(* Logix 5000 project; controller RG_Chopper vendor 1 type 14 code 235 rev 32.12; software revision 32.04; part 5 of 6 *)
(* tags used below, declared in another part *)
   CIP_CAUSTIC_RUNNING : ALIAS FOR SIGNAL_OUT_RG_CHOPPER.4;
   CYC_RUN : BOOL;   // Production Cycle Running
   DBX102_CTL : HOA_CTRL_v2;   // DBX102 Product Discharge Pump Control Block
   DBX102_FAULT : BOOL;   // DBX-102 Discharge Pump Drive Fault
   DBX102_M_FAULT : BOOL;   // DBX-102 Discharge Pump Drive or Motor Fault
   DBX102_SPD : ANLG_SCALE;   // DBX-102 Product Pump Speed Scaling
   DBX102_SPD_AM : PUSH_PUSH_PB;   // DBX-102 Speed Push-Push Button Control
   DBX102_SPD_IN : REAL;   // DBX-102 Product Pump User Requested Speed
   DBX102_SPD_OUT : REAL;   // DBX-102 VFD Alternate Requested Speed
   DBX102_SPD_PB : BOOL;   // DBX-102 Speed Auto / Manual PB
   DBX102_SPD_REQ : REAL;   // DBX-102 VFD Requested Speed
   DBX102_START : BOOL;   // DBX-102 Product Pump VFD START
   DBX102B_S_En : BOOL;   // DBX-102 Drive Safety Enable
   DBX103_AUX : BOOL;   // DBX-103 Water Pump Aux
   DBX104_CTL : HOA_CTRL_v2;   // DBX-104 Reversing Motor Starter Control
   DBX104_DWN : BOOL;   // DBX-104 Drum Dumper VFD Direction DOWN
   DBX104_FAULT : BOOL;   // DBX-104 Dumper Elevator Drive Fault
   DBX104_M_FAULT : BOOL;   // DBX-104 Dumper Elevator Drive or Motor Fault
   DBX104_S_DIR_EN : BOOL;   // DBX-104 Dump Elevator Direction Enabled
   DBX104_S_DWN : BOOL;   // DBX-104 Dump Elevator DOWN (Safety)
   DBX104_S_START : BOOL;   // DBX-104 Dump Elevator START (Safety)
   DBX104_S_UP : BOOL;   // DBX-104 Dump Elevator UP (Safety)
   DBX104_SPD : ANLG_SCALE;   // DBX-104 Product Pump Speed Scaling
   DBX104_SPD_AM : PUSH_PUSH_PB;   // DBX-104 Speed Push-Push Button Control
   DBX104_SPD_IN : DINT;   // DBX-102 Product Pump User Requested Speed
   DBX104_SPD_OUT : DINT;   // DBX-104 VFD Alternate Requested Speed
   DBX104_SPD_PB : BOOL;   // DBX-104 Speed Auto / Manual PB
   DBX104_SPD_REQ : DINT;   // DBX-104 VFD Requested Speed
   DBX104_START : BOOL;   // DBX-104 Drum Dumper VFD START
   DBX104_UP : BOOL;   // DBX-104 Drum Dumper VFD Direction UP
   DBX104B_S_En : BOOL;   // DBX-104 Drive Enable Safety
   DL101_Scl : REAL;
   DLT101_LVL_SCL : REAL;   // Tank Level Scaled (0.0 - 100.0%)
   DLT101_Tk : TK_CTRL;   // Tank Level Control
   DTT101 : REAL;   // DTT-101 Hot Water Temperature Analong In
   DWN_MKBK : BOOL;   // Elevator Down Make / Break LS_L1 Detection
   Fault_ACK : BOOL;   // Fault Acknowledge
   Gate_SW1 : DCI_MONITOR;   // Safety Switch Gate_SW1 SW105 A/B
   Gate_SW2 : DCI_MONITOR;   // Safety Switch Gate_SW2 SW108 A/B
   HMI_FLT_RES : BOOL;   // Safety Module Fault Reset HMI
   HT_TEMP_SP : REAL;   // TCV-101 SetPoint from HMI
   ILG104_GREEN_STACK : BOOL;   // Stack Light Green
   ILG105_YELLOW_STACK : BOOL;   // Stack Light Yellow
   ILG106_RED_STACK : BOOL;   // Stack Light Red
   KR101_DUMPER_PERM : BOOL;   // Dumper Permissive NON-FATAL ALARM 0 = ALARM
   LEVEL_TIMER : TIMER;   // Juice Tank At High Level
   LSS_LOT1 : BOOL;   // New Dumper LOWER OVER TRAVEL Limit Switch
   M104S_DWN_CTL : CONFIGURABLE_ROUT;   // DBX-104 Dump Elevator Safety Starter Down Output
   M104S_STRT_CTL : CONFIGURABLE_ROUT;   // DBX-104 Dump Elevator Safety Starter Enable Output
   M104S_UP_CTL : CONFIGURABLE_ROUT;   // DBX-104 Dump Elevator Safety Starter UP Output
   ONESHOT : DINT;   // One-shot Word
   S_ESTOP : BOOL;   // Safety ESTOP
   S_ESTOP_1 : EMERGENCY_STOP;   // Safety ESTOP Block #1
   S_ESTOP_2 : EMERGENCY_STOP;   // Safety ESTOP Block #2
   S_Fault_Res : BOOL;   // Safety Circuit Fault Reset
   S_SW_IN : DINT;   // Safety Switch Input Array
   SIGNAL_OUT_RG_CHOPPER : DINT;
   SPARE_OUT : DINT;
   ST_S_SW : DINT;   // Safety Switch Status Output Array
   SW106_LC : LIGHT_CURTAIN;   // Safety SW106 Light Curain
   Tank_Lid1 : EMERGENCY_STOP;   // Safety Switch Tank Lid Status SW105 A/B
   TCV101_AM : PUSH_PUSH_PB;   // TCV-101 Temperature Control Man / Auto Push-Push
   TCV101_AO : DINT;   // TCV-101 Temperature Control Valve Analog Out
   TCV101_Auto : BOOL;   // TCV-101 Temp Control Loop Auto
   TCV101_CTL : PID;   // PCV-101 PID Temperature Control
   TCV101_CTL_ST : DINT;   // TCV-101 Control Status 0= Auto 1= Manual 2= Error
   TCV101_Man : BOOL;   // TCV-101 Temp Control Loop Manual
   TCV101_PB : BOOL;   // TCV-101 Temperature Control Man / Auto PB
   TCV101_SP_MAX : REAL;   // TCV101 PID Max Temp SP
   TCV101_SP_MIN : REAL;   // PCV-101 PID Temp SP MIN
   UP_MKBK : BOOL;   // Elevator Down Make / Break LS_U1 Detection
   VALV_OUT : REAL;   // TCV-101 Temp Control Valve Pos Output
   WTR_HI_TEMP : BOOL;   // High Water Temperature Alarm
(* MainProgram, continued *)

ROUTINE OutLink   (* ladder *)
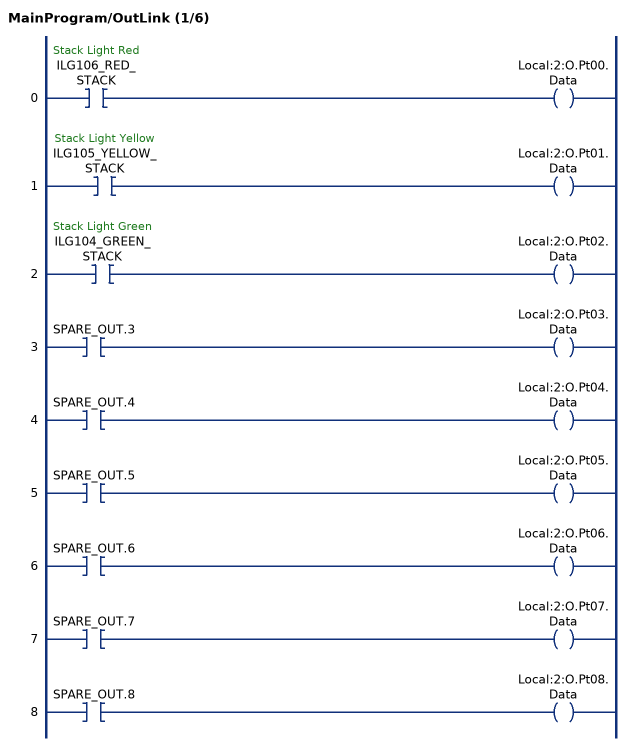
   0: XIC(ILG106_RED_STACK)OTE(Local:2:O.Pt00.Data);
   1: XIC(ILG105_YELLOW_STACK)OTE(Local:2:O.Pt01.Data);
   2: XIC(ILG104_GREEN_STACK)OTE(Local:2:O.Pt02.Data);
   3: XIC(SPARE_OUT.3)OTE(Local:2:O.Pt03.Data);
   4: XIC(SPARE_OUT.4)OTE(Local:2:O.Pt04.Data);
   5: XIC(SPARE_OUT.5)OTE(Local:2:O.Pt05.Data);
   6: XIC(SPARE_OUT.6)OTE(Local:2:O.Pt06.Data);
   7: XIC(SPARE_OUT.7)OTE(Local:2:O.Pt07.Data);
   8: XIC(SPARE_OUT.8)OTE(Local:2:O.Pt08.Data);
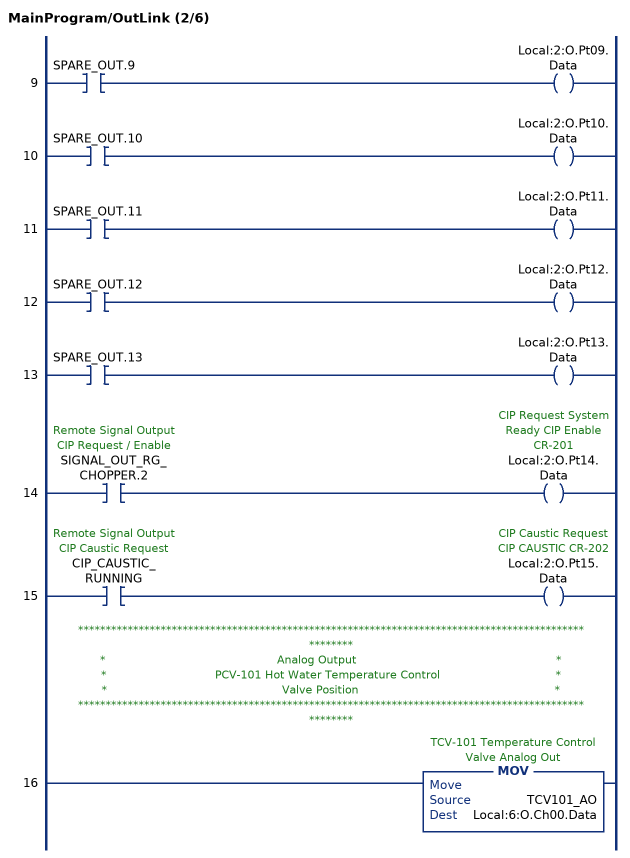
   9: XIC(SPARE_OUT.9)OTE(Local:2:O.Pt09.Data);
   10: XIC(SPARE_OUT.10)OTE(Local:2:O.Pt10.Data);
   11: XIC(SPARE_OUT.11)OTE(Local:2:O.Pt11.Data);
   12: XIC(SPARE_OUT.12)OTE(Local:2:O.Pt12.Data);
   13: XIC(SPARE_OUT.13)OTE(Local:2:O.Pt13.Data);
   14: XIC(SIGNAL_OUT_RG_CHOPPER.2)OTE(Local:2:O.Pt14.Data);
   15: XIC(CIP_CAUSTIC_RUNNING)OTE(Local:2:O.Pt15.Data);
   // ****************************************************************************************************
   // *                                                 Analog Output                                                         *
   // *                               PCV-101 Hot Water Temperature Control                                 *
   // *                                                  Valve Position                                                        *
   // ****************************************************************************************************
   16: MOV(TCV101_AO,Local:6:O.Ch00.Data);
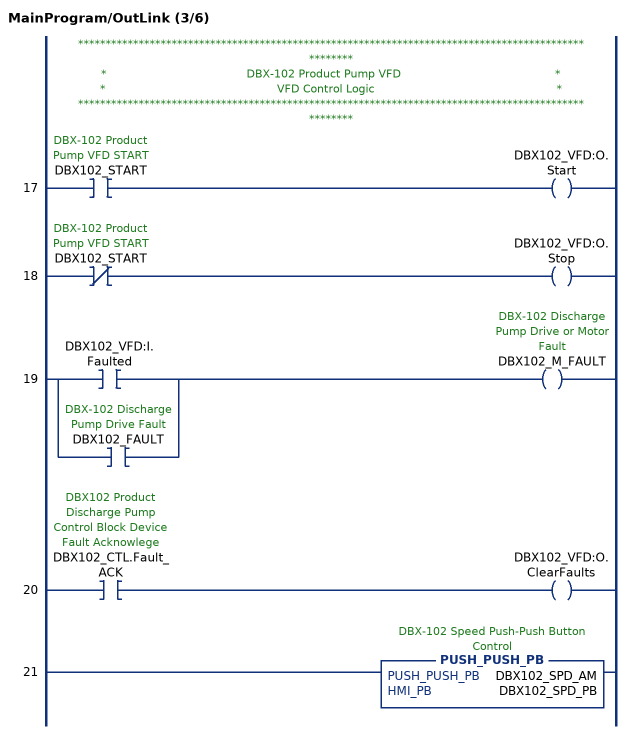
   // ****************************************************************************************************
   // *                                        DBX-102 Product Pump VFD                                            *
   // *                                                 VFD Control Logic                                                    *
   // ****************************************************************************************************
   17: XIC(DBX102_START)OTE(DBX102_VFD:O.Start);
   18: XIO(DBX102_START)OTE(DBX102_VFD:O.Stop);
   19: [XIC(DBX102_VFD:I.Faulted) ,XIC(DBX102_FAULT) ]OTE(DBX102_M_FAULT);
   20: XIC(DBX102_CTL.Fault_ACK)OTE(DBX102_VFD:O.ClearFaults);
   21: PUSH_PUSH_PB(DBX102_SPD_AM,DBX102_SPD_PB);
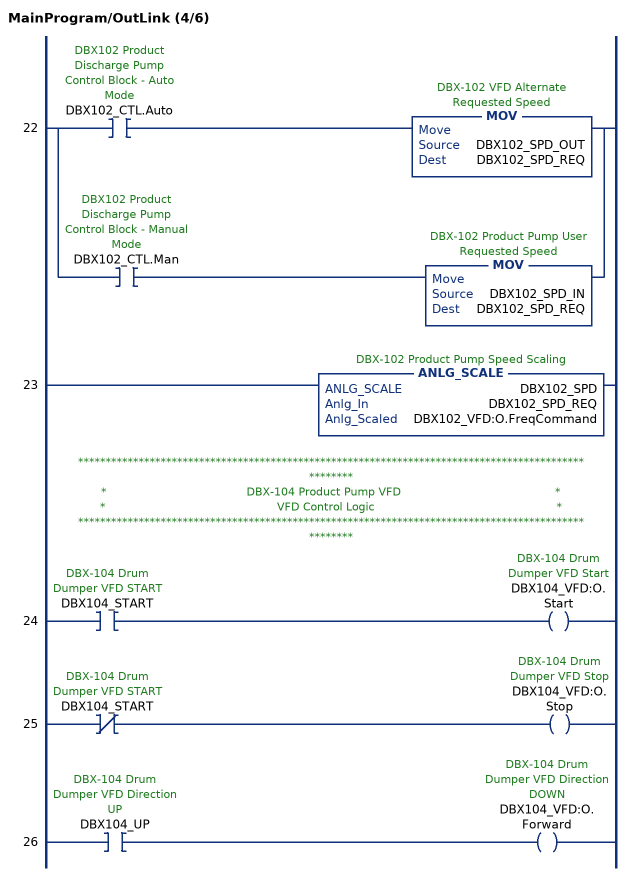
   22: [XIC(DBX102_CTL.Auto) MOV(DBX102_SPD_OUT,DBX102_SPD_REQ) ,XIC(DBX102_CTL.Man) MOV(DBX102_SPD_IN,DBX102_SPD_REQ) ];
   23: ANLG_SCALE(DBX102_SPD,DBX102_SPD_REQ,DBX102_VFD:O.FreqCommand);
   // ****************************************************************************************************
   // *                                        DBX-104 Product Pump VFD                                            *
   // *                                                 VFD Control Logic                                                    *
   // ****************************************************************************************************
   24: XIC(DBX104_START)OTE(DBX104_VFD:O.Start);
   25: XIO(DBX104_START)OTE(DBX104_VFD:O.Stop);
   26: XIC(DBX104_UP)OTE(DBX104_VFD:O.Forward);
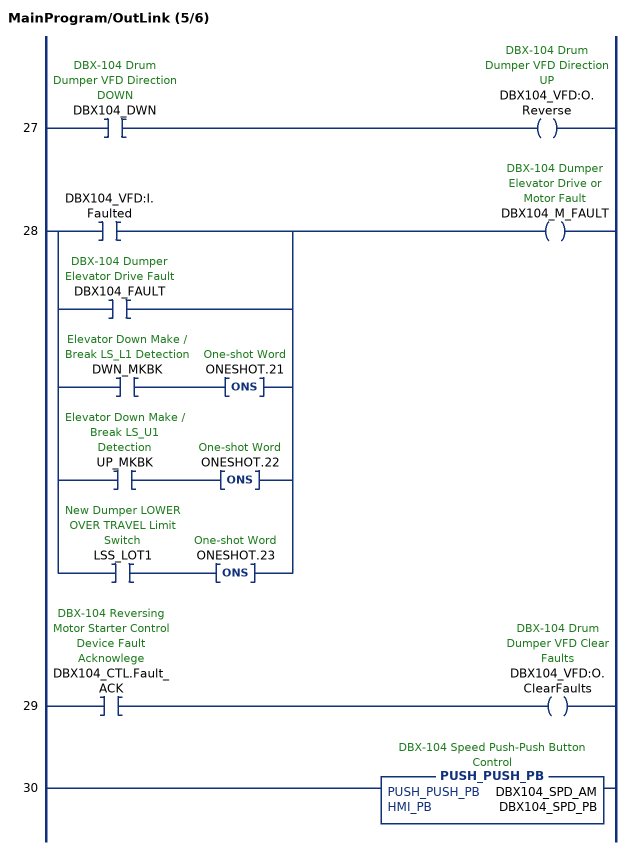
   27: XIC(DBX104_DWN)OTE(DBX104_VFD:O.Reverse);
   28: [XIC(DBX104_VFD:I.Faulted) ,XIC(DBX104_FAULT) ,XIC(DWN_MKBK) ONS(ONESHOT.21) ,XIC(UP_MKBK) ONS(ONESHOT.22) ,XIC(LSS_LOT1) ONS(ONESHOT.23) ]OTE(DBX104_M_FAULT);
   29: XIC(DBX104_CTL.Fault_ACK)OTE(DBX104_VFD:O.ClearFaults);
   30: PUSH_PUSH_PB(DBX104_SPD_AM,DBX104_SPD_PB);
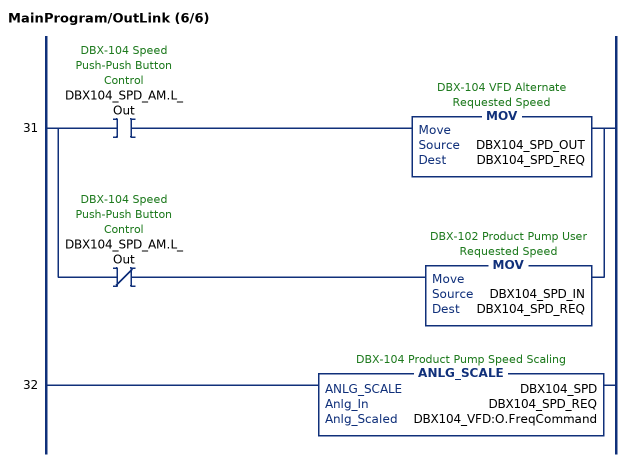
   31: [XIC(DBX104_SPD_AM.L_Out) MOV(DBX104_SPD_OUT,DBX104_SPD_REQ) ,XIO(DBX104_SPD_AM.L_Out) MOV(DBX104_SPD_IN,DBX104_SPD_REQ) ];
   32: ANLG_SCALE(DBX104_SPD,DBX104_SPD_REQ,DBX104_VFD:O.FreqCommand);
END_ROUTINE

ROUTINE TANK_LVL   (* ladder *)
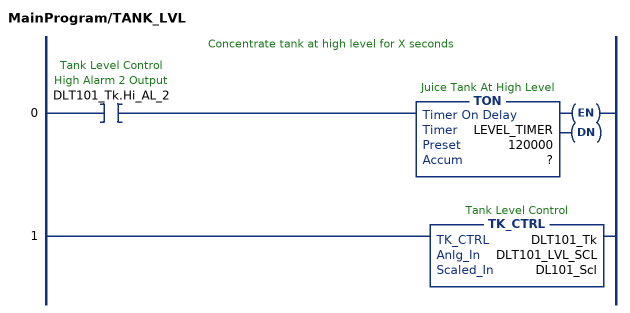
   // Concentrate tank at high level for X seconds
   0: XIC(DLT101_Tk.Hi_AL_2)TON(LEVEL_TIMER,?,?);
   1: TK_CTRL(DLT101_Tk,DLT101_LVL_SCL,DL101_Scl);
END_ROUTINE

ROUTINE TEMP_CTRL   (* ladder *)
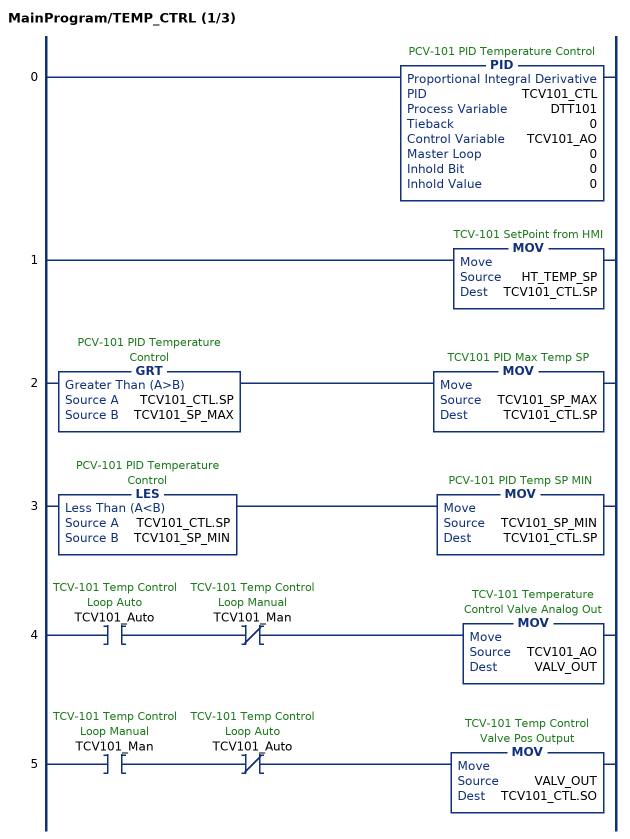
   0: PID(TCV101_CTL,DTT101,0,TCV101_AO,0,0,0);
   1: MOV(HT_TEMP_SP,TCV101_CTL.SP);
   2: GRT(TCV101_CTL.SP,TCV101_SP_MAX)MOV(TCV101_SP_MAX,TCV101_CTL.SP);
   3: LES(TCV101_CTL.SP,TCV101_SP_MIN)MOV(TCV101_SP_MIN,TCV101_CTL.SP);
   4: XIC(TCV101_Auto)XIO(TCV101_Man)MOV(TCV101_AO,VALV_OUT);
   5: XIC(TCV101_Man)XIO(TCV101_Auto)MOV(VALV_OUT,TCV101_CTL.SO);
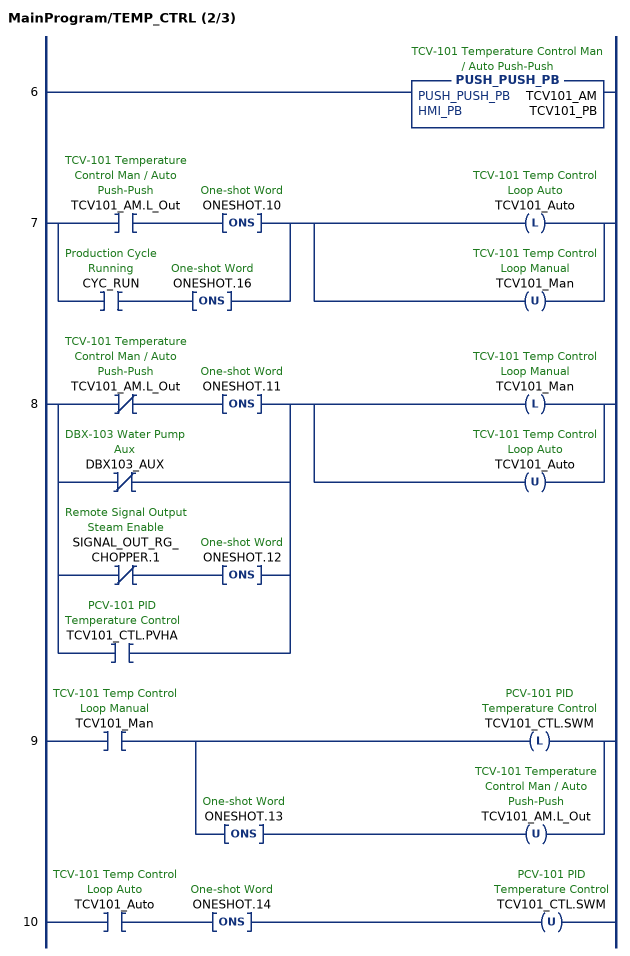
   6: PUSH_PUSH_PB(TCV101_AM,TCV101_PB);
   7: [XIC(TCV101_AM.L_Out) ONS(ONESHOT.10) ,XIC(CYC_RUN) ONS(ONESHOT.16) ][OTL(TCV101_Auto) ,OTU(TCV101_Man) ];
   8: [XIO(TCV101_AM.L_Out) ONS(ONESHOT.11) ,XIO(DBX103_AUX) ,XIO(SIGNAL_OUT_RG_CHOPPER.1) ONS(ONESHOT.12) ,XIC(TCV101_CTL.PVHA) ][OTL(TCV101_Man) ,OTU(TCV101_Auto) ];
   9: XIC(TCV101_Man)[OTL(TCV101_CTL.SWM) ,ONS(ONESHOT.13) OTU(TCV101_AM.L_Out) ];
   10: XIC(TCV101_Auto)ONS(ONESHOT.14)OTU(TCV101_CTL.SWM);
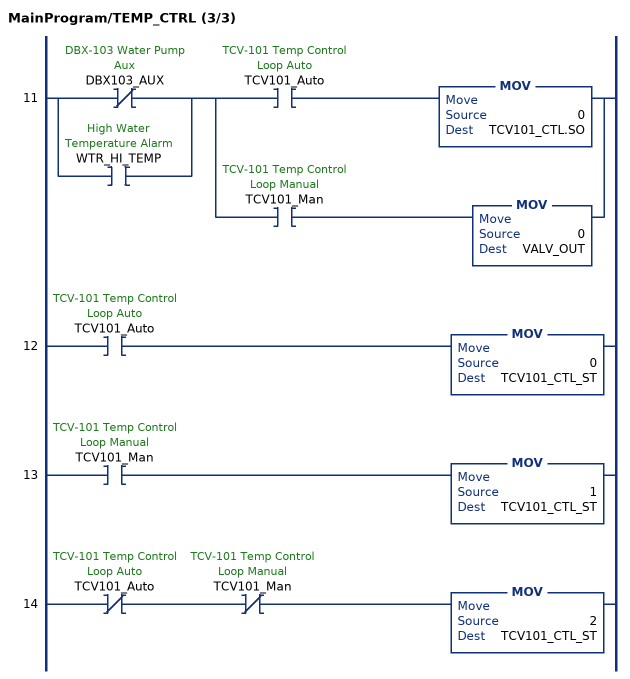
   11: [XIO(DBX103_AUX) ,XIC(WTR_HI_TEMP) ][XIC(TCV101_Auto) MOV(0,TCV101_CTL.SO) ,XIC(TCV101_Man) MOV(0,VALV_OUT) ];
   12: XIC(TCV101_Auto)MOV(0,TCV101_CTL_ST);
   13: XIC(TCV101_Man)MOV(1,TCV101_CTL_ST);
   14: XIO(TCV101_Auto)XIO(TCV101_Man)MOV(2,TCV101_CTL_ST);
END_ROUTINE
END_PROGRAM

PROGRAM SafetyProgram   (* main routine MainRoutine, safety *)

ROUTINE InLink   (* ladder *)
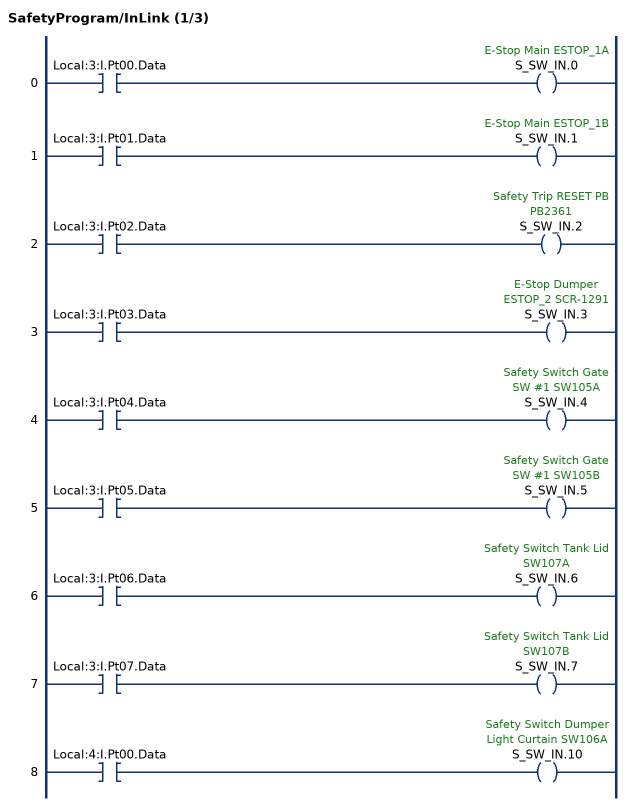
   0: XIC(Local:3:I.Pt00.Data)OTE(S_SW_IN.0);
   1: XIC(Local:3:I.Pt01.Data)OTE(S_SW_IN.1);
   2: XIC(Local:3:I.Pt02.Data)OTE(S_SW_IN.2);
   3: XIC(Local:3:I.Pt03.Data)OTE(S_SW_IN.3);
   4: XIC(Local:3:I.Pt04.Data)OTE(S_SW_IN.4);
   5: XIC(Local:3:I.Pt05.Data)OTE(S_SW_IN.5);
   6: XIC(Local:3:I.Pt06.Data)OTE(S_SW_IN.6);
   7: XIC(Local:3:I.Pt07.Data)OTE(S_SW_IN.7);
   8: XIC(Local:4:I.Pt00.Data)OTE(S_SW_IN.10);
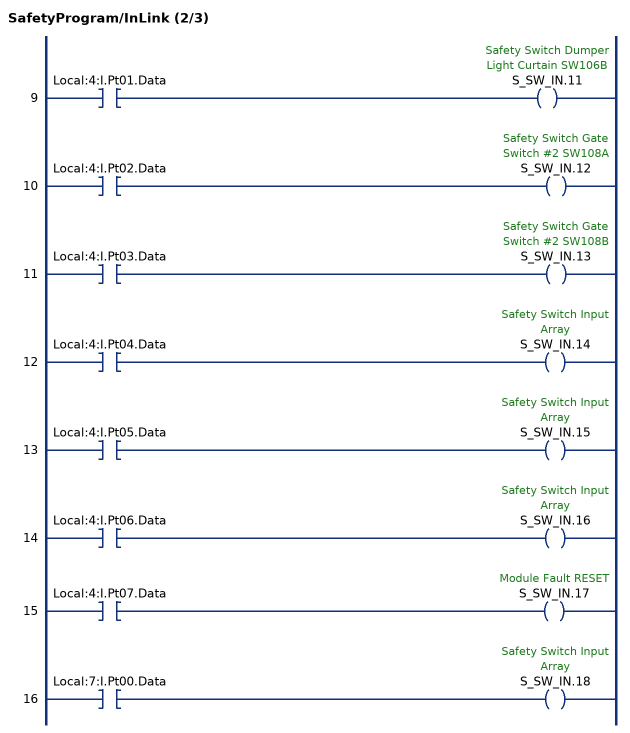
   9: XIC(Local:4:I.Pt01.Data)OTE(S_SW_IN.11);
   10: XIC(Local:4:I.Pt02.Data)OTE(S_SW_IN.12);
   11: XIC(Local:4:I.Pt03.Data)OTE(S_SW_IN.13);
   12: XIC(Local:4:I.Pt04.Data)OTE(S_SW_IN.14);
   13: XIC(Local:4:I.Pt05.Data)OTE(S_SW_IN.15);
   14: XIC(Local:4:I.Pt06.Data)OTE(S_SW_IN.16);
   15: XIC(Local:4:I.Pt07.Data)OTE(S_SW_IN.17);
   16: XIC(Local:7:I.Pt00.Data)OTE(S_SW_IN.18);
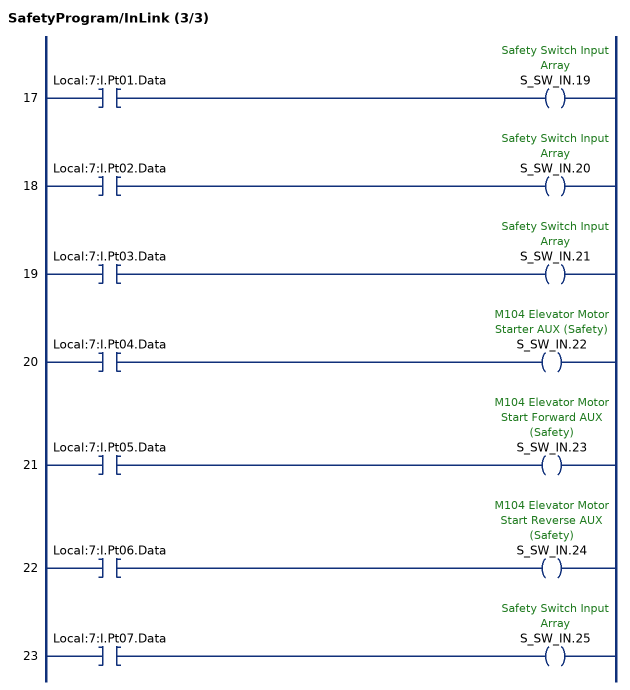
   17: XIC(Local:7:I.Pt01.Data)OTE(S_SW_IN.19);
   18: XIC(Local:7:I.Pt02.Data)OTE(S_SW_IN.20);
   19: XIC(Local:7:I.Pt03.Data)OTE(S_SW_IN.21);
   20: XIC(Local:7:I.Pt04.Data)OTE(S_SW_IN.22);
   21: XIC(Local:7:I.Pt05.Data)OTE(S_SW_IN.23);
   22: XIC(Local:7:I.Pt06.Data)OTE(S_SW_IN.24);
   23: XIC(Local:7:I.Pt07.Data)OTE(S_SW_IN.25);
END_ROUTINE

ROUTINE LOGIC   (* ladder *)
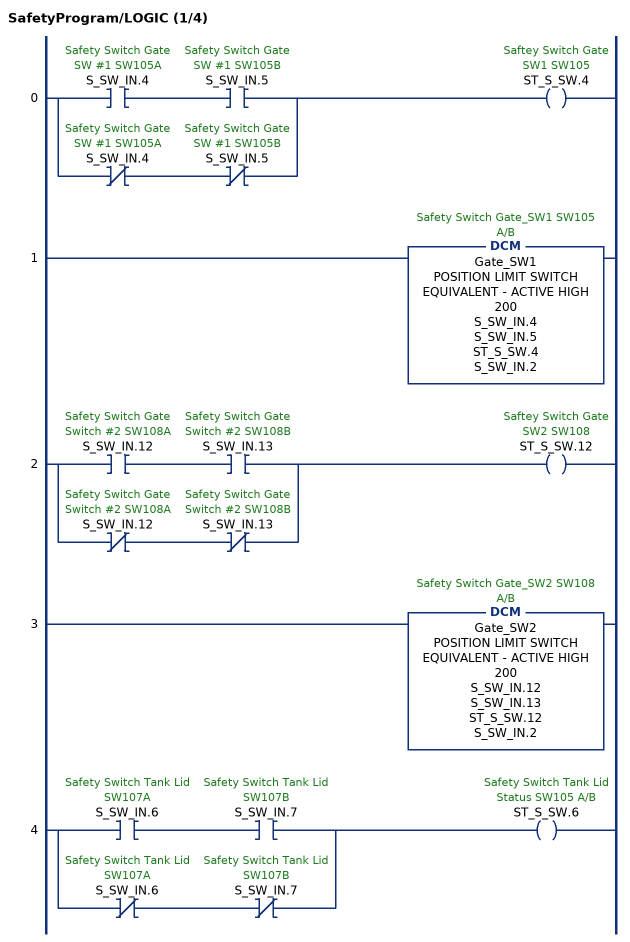
   0: [XIC(S_SW_IN.4) XIC(S_SW_IN.5) ,XIO(S_SW_IN.4) XIO(S_SW_IN.5) ]OTE(ST_S_SW.4);
   1: DCM(Gate_SW1,POSITION LIMIT SWITCH,EQUIVALENT - ACTIVE HIGH,200,S_SW_IN.4,S_SW_IN.5,ST_S_SW.4,S_SW_IN.2);
   2: [XIC(S_SW_IN.12) XIC(S_SW_IN.13) ,XIO(S_SW_IN.12) XIO(S_SW_IN.13) ]OTE(ST_S_SW.12);
   3: DCM(Gate_SW2,POSITION LIMIT SWITCH,EQUIVALENT - ACTIVE HIGH,200,S_SW_IN.12,S_SW_IN.13,ST_S_SW.12,S_SW_IN.2);
   4: [XIC(S_SW_IN.6) XIC(S_SW_IN.7) ,XIO(S_SW_IN.6) XIO(S_SW_IN.7) ]OTE(ST_S_SW.6);
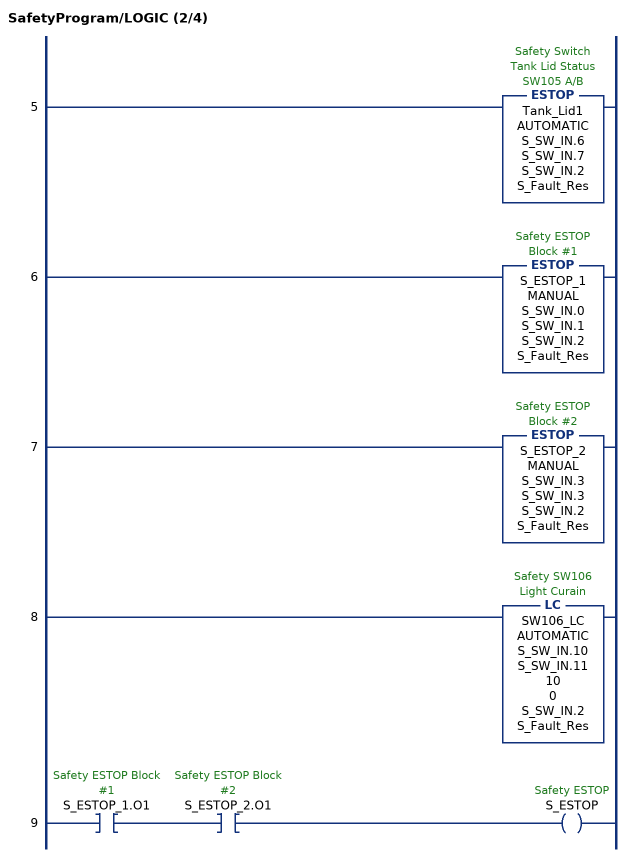
   5: ESTOP(Tank_Lid1,AUTOMATIC,S_SW_IN.6,S_SW_IN.7,S_SW_IN.2,S_Fault_Res);
   6: ESTOP(S_ESTOP_1,MANUAL,S_SW_IN.0,S_SW_IN.1,S_SW_IN.2,S_Fault_Res);
   7: ESTOP(S_ESTOP_2,MANUAL,S_SW_IN.3,S_SW_IN.3,S_SW_IN.2,S_Fault_Res);
   8: LC(SW106_LC,AUTOMATIC,S_SW_IN.10,S_SW_IN.11,10,0,S_SW_IN.2,S_Fault_Res);
   9: XIC(S_ESTOP_1.O1)XIC(S_ESTOP_2.O1)OTE(S_ESTOP);
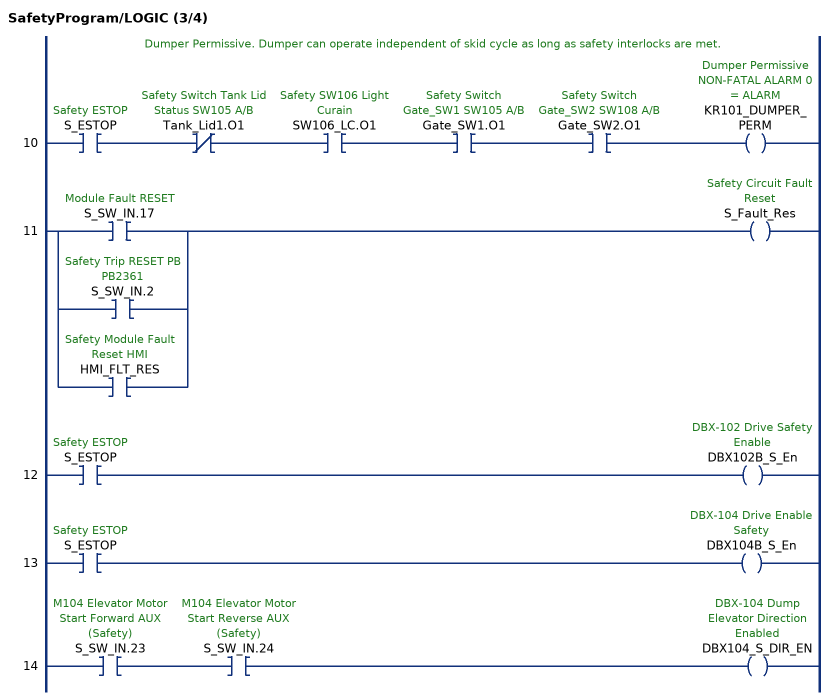
   // Dumper Permissive. Dumper can operate independent of skid cycle as long as safety interlocks are met.
   10: XIC(S_ESTOP)XIO(Tank_Lid1.O1)XIC(SW106_LC.O1)XIC(Gate_SW1.O1)XIC(Gate_SW2.O1)OTE(KR101_DUMPER_PERM);
   11: [XIC(S_SW_IN.17) ,XIC(S_SW_IN.2) ,XIC(HMI_FLT_RES) ]OTE(S_Fault_Res);
   12: XIC(S_ESTOP)OTE(DBX102B_S_En);
   13: XIC(S_ESTOP)OTE(DBX104B_S_En);
   14: XIC(S_SW_IN.23)XIC(S_SW_IN.24)OTE(DBX104_S_DIR_EN);
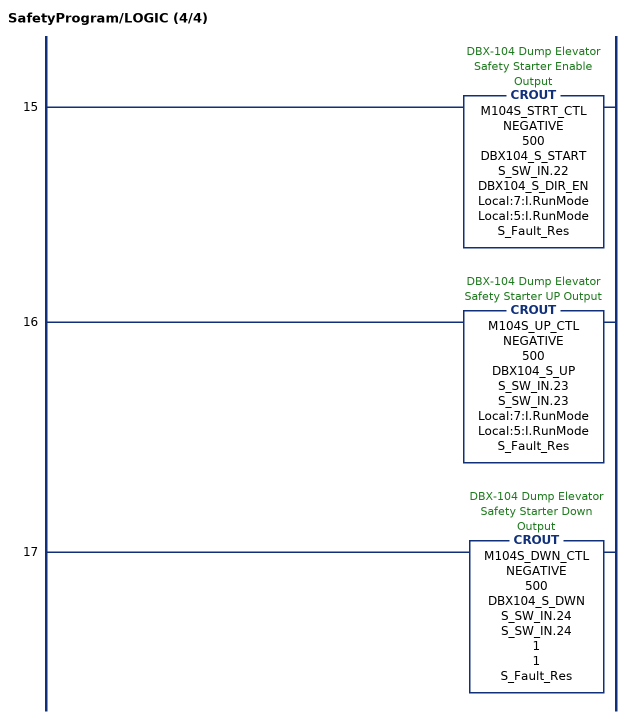
   15: CROUT(M104S_STRT_CTL,NEGATIVE,500,DBX104_S_START,S_SW_IN.22,DBX104_S_DIR_EN,Local:7:I.RunMode,Local:5:I.RunMode,S_Fault_Res);
   16: CROUT(M104S_UP_CTL,NEGATIVE,500,DBX104_S_UP,S_SW_IN.23,S_SW_IN.23,Local:7:I.RunMode,Local:5:I.RunMode,S_Fault_Res);
   17: CROUT(M104S_DWN_CTL,NEGATIVE,500,DBX104_S_DWN,S_SW_IN.24,S_SW_IN.24,1,1,S_Fault_Res);
END_ROUTINE

ROUTINE MainRoutine   (* ladder *)
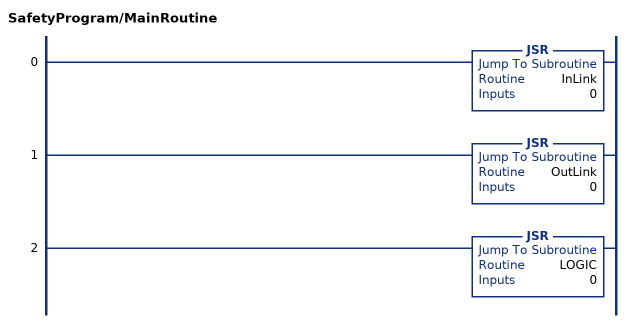
   0: JSR(InLink,0);
   1: JSR(OutLink,0);
   2: JSR(LOGIC,0);
END_ROUTINE
